// TIA Portal project "plc-automatic-manual-tank-level-control-pid" (V16)
// Vorlageprojekt für das Buch mit Zielsystem S7-1200

(* hardware
DEVICE "S7-1200-Station_1"  S7-1200 Station
   slot 0: "Baugruppenträger_0"  Rack  V1.0
   slot 1: "PLC_1"  CPU 1214C DC/DC/DC  6ES7 214-1AG40-0XB0  V4.4
   slot 2: "AQ 4x14BIT_1"  6ES7 232-4HD32-0XB0  V2.1
DEVICE "HMI_1"  KTP700 Basic PN
   slot 0: "HMI_1"  KTP700 Basic PN  6AV2 123-2GB03-0AX0  16.0.0.0
   slot 1: "HMI_RT_1"  KTP700 Basic PN  6AV2 123-2GB03-0AX0  16.0.0.0
   slot 5: "HMI_1.IE_CP_1"  PROFINET Interface  16.0.0.0
      slot 1: "PROFINET Interface_1"  PROFINET Interface
         slot 1: "Port_1"  Port
*)

// ===== PLC "PLC_1"  CPU 1214C DC/DC/DC =====

VAR_GLOBAL   // PLC tag table "Standard-Variablentabelle"
   "Seviye_Sensörü" AT %IW30 : Int;
   "Doldurma_Valfi" AT %QW30 : Int;
   "Set_Point" AT %MW32 : Int;
   "HMI_Doldurma_But" AT %M5.0 : Bool;
   "PID_Çıkış_Mem" AT %MW10 : Int;
   "HMI_OTO_MAN" AT %M5.1 : Bool;
   "HMI_Boşaltma_But" AT %M5.3 : Bool;
   "Man_Doldurma_Mem" AT %M5.4 : Bool;
   "DolVlf_Açıklık_DInt" AT %MD12 : DInt;
   "Otomatik_Start_Mem" AT %M5.5 : Bool;
   "HMI_Sıvı_Seviye" AT %MD34 : Real;
   "DolVlf_Açıklık_Yüzde_DInt" AT %MD16 : DInt;
   "Sıvı_Seviye_Mem" AT %MW38 : Int;
   "Sıvı_Seviye" AT %MD40 : Real;
   "Boşaltma_Valfi" AT %QW32 : Int;
   "Üst_Limit" AT %M5.7 : Bool;
   "Man_Boşaltma_Mem" AT %M6.0 : Bool;
   "HMI_DolVlf_Açıklık_Arttır_But" AT %M6.1 : Bool;
   "HMI_DolVlf_Açıklık_Azalt_But" AT %M6.2 : Bool;
   "HMI_BoşVlf_Açıklık_Arttır_But" AT %M6.3 : Bool;
   "HMI_BoşVlf_Açıklık_Azalt_But" AT %M6.4 : Bool;
   "DolVlf_Açıklık_Mem" AT %MW44 : Int;
   "BoşVlf_Açıklık_Mem" AT %MW46 : Int;
   "HMI_DolVlf_Açıklık_Yüzde" AT %MW20 : Int;
   "BoşVlf_Açıklık_DInt" AT %MD22 : DInt;
   "BoşVlf_Açıklık_Yüzde_DInt" AT %MD26 : DInt;
   "HMI_BoşVlf_Açıklık_Yüzde" AT %MW30 : Int;
   "Kenar_Tetikleme_1" AT %M6.5 : Bool;
   "Kenar_Tetikleme_2" AT %M6.6 : Bool;
   "Kenar_Tetikleme_3" AT %M6.7 : Bool;
   "Kenar_Tetikleme_4" AT %M7.0 : Bool;
   "DolVlf_Açıklık_Kontrol" AT %MW50 : Int;
   "HMI_Stop_But" AT %M5.2 : Bool;
   "Clock_Byte" AT %MB0 : Byte;
   "Clock_10Hz" AT %M0.0 : Bool;
   "Clock_5Hz" AT %M0.1 : Bool;
   "Clock_2.5Hz" AT %M0.2 : Bool;
   "Clock_2Hz" AT %M0.3 : Bool;
   "Clock_1.25Hz" AT %M0.4 : Bool;
   "Clock_1Hz" AT %M0.5 : Bool;
   "Clock_0.625Hz" AT %M0.6 : Bool;
   "Clock_0.5Hz" AT %M0.7 : Bool;
   "Stop_Uyarı" AT %M7.1 : Bool;
END_VAR

FUNCTION "Manuel_Çalışma" : Void   // FC1, LAD
{ S7_Optimized_Access := 'TRUE' }
VERSION : 0.1
BEGIN

REGION Network 1
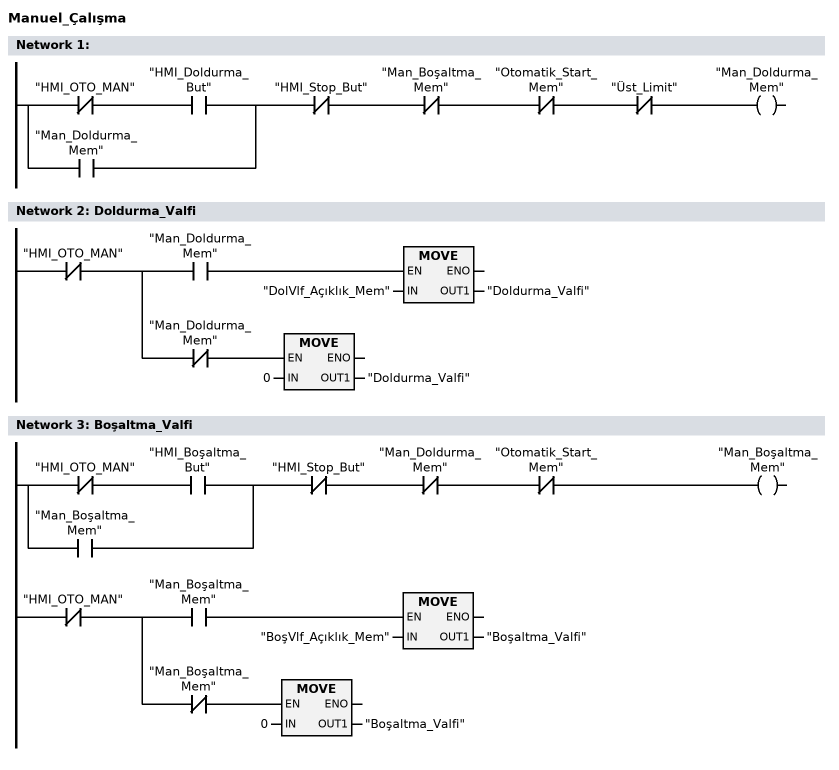
   RUNG wire#powerrail
      I_Contact( "HMI_OTO_MAN" )
      Contact( "HMI_Doldurma_But" )
      wire#w1
      I_Contact( "HMI_Stop_But" )
      I_Contact( "Man_Boşaltma_Mem" )
      I_Contact( "Otomatik_Start_Mem" )
      I_Contact( "Üst_Limit" )
      Coil( "Man_Doldurma_Mem" )
   END_RUNG
   RUNG wire#powerrail
      Contact( "Man_Doldurma_Mem" )
   END_RUNG wire#w1
   // the same network as SCL:
   "Man_Doldurma_Mem" := ((NOT "HMI_OTO_MAN" AND "HMI_Doldurma_But") OR "Man_Doldurma_Mem") AND NOT "HMI_Stop_But" AND NOT "Man_Boşaltma_Mem" AND NOT "Otomatik_Start_Mem" AND NOT "Üst_Limit";
END_REGION

REGION Network 2: Doldurma_Valfi
   RUNG wire#powerrail
      I_Contact( "HMI_OTO_MAN" )
      wire#w1
      Contact( "Man_Doldurma_Mem" )
      Move(in := "DolVlf_Açıklık_Mem", out1 => "Doldurma_Valfi")
   END_RUNG
   RUNG wire#w1
      I_Contact( "Man_Doldurma_Mem" )
      Move(in := 0, out1 => "Doldurma_Valfi")
   END_RUNG
   // the same network as SCL:
   IF NOT "HMI_OTO_MAN" AND "Man_Doldurma_Mem" THEN "Doldurma_Valfi" := "DolVlf_Açıklık_Mem"; END_IF;
   IF NOT "HMI_OTO_MAN" AND NOT "Man_Doldurma_Mem" THEN "Doldurma_Valfi" := 0; END_IF;
END_REGION

REGION Network 3: Boşaltma_Valfi
   RUNG wire#powerrail
      I_Contact( "HMI_OTO_MAN" )
      Contact( "HMI_Boşaltma_But" )
      wire#w1
      I_Contact( "HMI_Stop_But" )
      I_Contact( "Man_Doldurma_Mem" )
      I_Contact( "Otomatik_Start_Mem" )
      Coil( "Man_Boşaltma_Mem" )
   END_RUNG
   RUNG wire#powerrail
      Contact( "Man_Boşaltma_Mem" )
   END_RUNG wire#w1
   RUNG wire#powerrail
      I_Contact( "HMI_OTO_MAN" )
      wire#w2
      Contact( "Man_Boşaltma_Mem" )
      Move(in := "BoşVlf_Açıklık_Mem", out1 => "Boşaltma_Valfi")
   END_RUNG
   RUNG wire#w2
      I_Contact( "Man_Boşaltma_Mem" )
      Move(in := 0, out1 => "Boşaltma_Valfi")
   END_RUNG
   // the same network as SCL:
   "Man_Boşaltma_Mem" := ((NOT "HMI_OTO_MAN" AND "HMI_Boşaltma_But") OR "Man_Boşaltma_Mem") AND NOT "HMI_Stop_But" AND NOT "Man_Doldurma_Mem" AND NOT "Otomatik_Start_Mem";
   IF NOT "HMI_OTO_MAN" AND "Man_Boşaltma_Mem" THEN "Boşaltma_Valfi" := "BoşVlf_Açıklık_Mem"; END_IF;
   IF NOT "HMI_OTO_MAN" AND NOT "Man_Boşaltma_Mem" THEN "Boşaltma_Valfi" := 0; END_IF;
END_REGION
END_FUNCTION

FUNCTION "Otomatik_Çalışma" : Void   // FC2, LAD
{ S7_Optimized_Access := 'TRUE' }
VERSION : 0.1
BEGIN

REGION Network 1
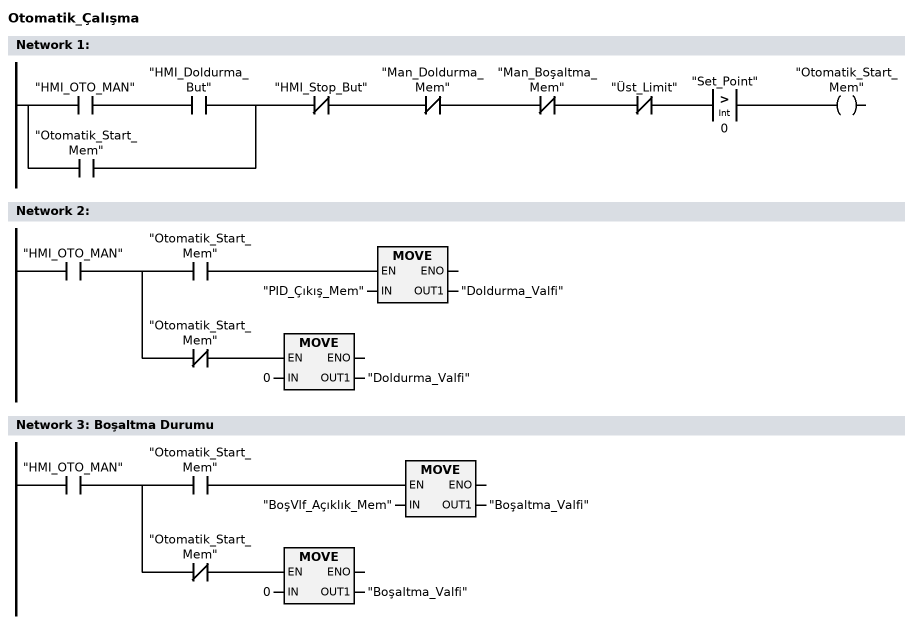
   RUNG wire#powerrail
      Contact( "HMI_OTO_MAN" )
      Contact( "HMI_Doldurma_But" )
      wire#w1
      I_Contact( "HMI_Stop_But" )
      I_Contact( "Man_Doldurma_Mem" )
      I_Contact( "Man_Boşaltma_Mem" )
      I_Contact( "Üst_Limit" )
      { S7_Templates := "SrcType := Int" } GT_Contact(in1 := "Set_Point", in2 := 0)
      Coil( "Otomatik_Start_Mem" )
   END_RUNG
   RUNG wire#powerrail
      Contact( "Otomatik_Start_Mem" )
   END_RUNG wire#w1
   // the same network as SCL:
   "Otomatik_Start_Mem" := (("HMI_OTO_MAN" AND "HMI_Doldurma_But") OR "Otomatik_Start_Mem") AND NOT "HMI_Stop_But" AND NOT "Man_Doldurma_Mem" AND NOT "Man_Boşaltma_Mem" AND NOT "Üst_Limit" AND ("Set_Point" > 0);
END_REGION

REGION Network 2
   RUNG wire#powerrail
      Contact( "HMI_OTO_MAN" )
      wire#w1
      Contact( "Otomatik_Start_Mem" )
      Move(in := "PID_Çıkış_Mem", out1 => "Doldurma_Valfi")
   END_RUNG
   RUNG wire#w1
      I_Contact( "Otomatik_Start_Mem" )
      Move(in := 0, out1 => "Doldurma_Valfi")
   END_RUNG
   // the same network as SCL:
   IF "HMI_OTO_MAN" AND "Otomatik_Start_Mem" THEN "Doldurma_Valfi" := "PID_Çıkış_Mem"; END_IF;
   IF "HMI_OTO_MAN" AND NOT "Otomatik_Start_Mem" THEN "Doldurma_Valfi" := 0; END_IF;
END_REGION

REGION Network 3: Boşaltma Durumu
   RUNG wire#powerrail
      Contact( "HMI_OTO_MAN" )
      wire#w1
      Contact( "Otomatik_Start_Mem" )
      Move(in := "BoşVlf_Açıklık_Mem", out1 => "Boşaltma_Valfi")
   END_RUNG
   RUNG wire#w1
      I_Contact( "Otomatik_Start_Mem" )
      Move(in := 0, out1 => "Boşaltma_Valfi")
   END_RUNG
   // the same network as SCL:
   IF "HMI_OTO_MAN" AND "Otomatik_Start_Mem" THEN "Boşaltma_Valfi" := "BoşVlf_Açıklık_Mem"; END_IF;
   IF "HMI_OTO_MAN" AND NOT "Otomatik_Start_Mem" THEN "Boşaltma_Valfi" := 0; END_IF;
END_REGION
END_FUNCTION

FUNCTION "MHJ-PLC-Lab-Function-S71200" : Void   // FC9000, SCL
{ S7_Optimized_Access := 'TRUE' }
VERSION : 0.1
   VAR_TEMP
      rdTimeReturn : Int;
      outputTime : DTL;
      SyncVal : Byte;
      forVal : Int;
      forVal_2 : Int;
      Value : Byte;
   END_VAR
   VAR CONSTANT
      CompVal : Byte := 16#34;
      Value_01 : Byte := 16#11;
      Value_01_DW : DWord := 16#A165_D992;
      Value_02_DW : DWord := 16#58BE_4401;
   END_VAR
BEGIN

   #Value:=PEEK(area := 16#82,
        dbNumber := 0,
        byteOffset := 511);
   #Value := #Value + 1;

   POKE(area := 16#82,
        dbNumber := 0,
        byteOffset := 511,
        value := #Value);

   POKE(area:=16#81,
        dbNumber:=0,
        byteOffset:=1016,
        value:=#Value_01_DW);
   POKE(area := 16#81,
        dbNumber := 0,
        byteOffset := 1020,
        value := #Value_02_DW);

   POKE(area := 16#81,
        dbNumber := 0,
        byteOffset := 511,
        value := B#16#00);

   FOR #forVal := 0 TO 120 DO
       FOR #forVal_2:=0 TO 10 DO
           #rdTimeReturn:=RD_SYS_T(#outputTime);
           #rdTimeReturn := WR_SYS_T(#outputTime);
           #rdTimeReturn := RD_SYS_T(#outputTime);
           #rdTimeReturn := WR_SYS_T(#outputTime);
       END_FOR;
       #SyncVal:= PEEK(area := 16#81,
                      dbNumber := 0,
                      byteOffset := 511);
       IF #SyncVal = #CompVal THEN
          GOTO M_1;
       END_IF;
   END_FOR;
   RETURN;

   M_1:
   POKE(area := 16#81,
        dbNumber := 0,
        byteOffset := 511,
        value := B#16#0);
END_FUNCTION

ORGANIZATION_BLOCK "Main"   // OB1, LAD, ProgramCycle
TITLE = "Main Program Sweep (Cycle)"
{ S7_Optimized_Access := 'TRUE' }
VERSION : 0.1
   VAR_INPUT
      Initial_Call : Bool;   // Initial call of this OB
      Remanence : Bool;   // =True, if remanent data are available
   END_VAR
   VAR_TEMP   // added for the SCL form of the ladder/FBD networks
      _w1 : Bool;
      _w2 : Bool;
   END_VAR
BEGIN

REGION Network 1: Konnektierungsbaustein für PLC-Lab
   // Im Netzwerk 1 wird der Konnektierungsbaustein für PLC-Lab aufgerufen.
   // Dieser Aufruf darf nicht entfernt werden!
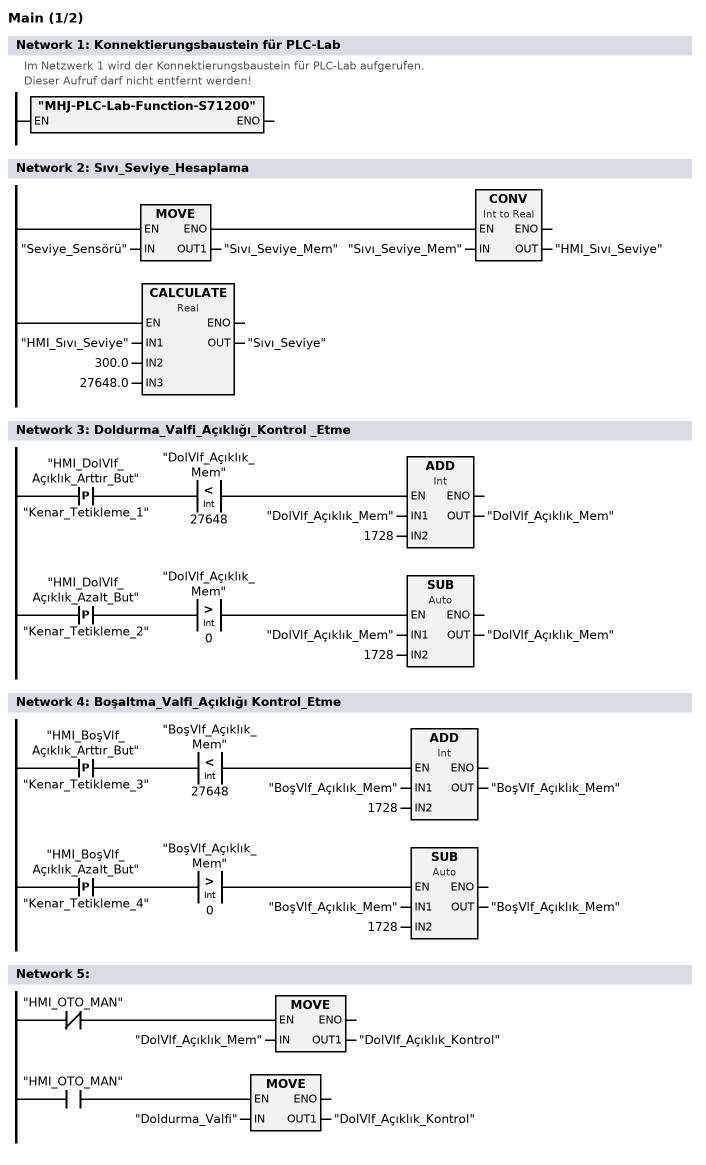
   RUNG wire#powerrail
      "MHJ-PLC-Lab-Function-S71200"()
   END_RUNG
   // the same network as SCL:
   "MHJ-PLC-Lab-Function-S71200"();
END_REGION

REGION Network 2: Sıvı_Seviye_Hesaplama
   RUNG wire#powerrail
      Move(in := "Seviye_Sensörü", out1 => "Sıvı_Seviye_Mem")
      { S7_Templates := "[SrcType := Int, DestType := Real]" } Convert(in := "Sıvı_Seviye_Mem", out => "HMI_Sıvı_Seviye")
   END_RUNG
   RUNG wire#powerrail
      { S7_Templates := "SrcType := Real"; S7_Expression := "(IN1*IN2)/IN3" } Calculate(in1 := "HMI_Sıvı_Seviye", in2 := 300.0, in3 := 27648.0, out => "Sıvı_Seviye")
   END_RUNG
   // the same network as SCL:
   "Sıvı_Seviye_Mem" := "Seviye_Sensörü";
   "HMI_Sıvı_Seviye" := INT_TO_REAL("Sıvı_Seviye_Mem");
   "Sıvı_Seviye" := ("HMI_Sıvı_Seviye"*300.0)/27648.0;
END_REGION

REGION Network 3: Doldurma_Valfi_Açıklığı_Kontrol _Etme
   RUNG wire#powerrail
      P_Contact(operand := "HMI_DolVlf_Açıklık_Arttır_But", bit := "Kenar_Tetikleme_1")
      { S7_Templates := "SrcType := Int" } LT_Contact(in1 := "DolVlf_Açıklık_Mem", in2 := 27648)
      { S7_Templates := "SrcType := Int" } Add(in1 := "DolVlf_Açıklık_Mem", in2 := 1728, out => "DolVlf_Açıklık_Mem")
   END_RUNG
   RUNG wire#powerrail
      P_Contact(operand := "HMI_DolVlf_Açıklık_Azalt_But", bit := "Kenar_Tetikleme_2")
      { S7_Templates := "SrcType := Int" } GT_Contact(in1 := "DolVlf_Açıklık_Mem", in2 := 0)
      Sub(in1 := "DolVlf_Açıklık_Mem", in2 := 1728, out => "DolVlf_Açıklık_Mem")
   END_RUNG
   // the same network as SCL:
   #_w1 := "HMI_DolVlf_Açıklık_Arttır_But" AND NOT "Kenar_Tetikleme_1";   // rising edge of "HMI_DolVlf_Açıklık_Arttır_But"
   "Kenar_Tetikleme_1" := "HMI_DolVlf_Açıklık_Arttır_But";
   IF #_w1 AND ("DolVlf_Açıklık_Mem" < 27648) THEN
       "DolVlf_Açıklık_Mem" := "DolVlf_Açıklık_Mem" + 1728;
   END_IF;
   #_w2 := "HMI_DolVlf_Açıklık_Azalt_But" AND NOT "Kenar_Tetikleme_2";   // rising edge of "HMI_DolVlf_Açıklık_Azalt_But"
   "Kenar_Tetikleme_2" := "HMI_DolVlf_Açıklık_Azalt_But";
   IF #_w2 AND ("DolVlf_Açıklık_Mem" > 0) THEN "DolVlf_Açıklık_Mem" := "DolVlf_Açıklık_Mem" - 1728; END_IF;
END_REGION

REGION Network 4: Boşaltma_Valfi_Açıklığı Kontrol_Etme
   RUNG wire#powerrail
      P_Contact(operand := "HMI_BoşVlf_Açıklık_Arttır_But", bit := "Kenar_Tetikleme_3")
      { S7_Templates := "SrcType := Int" } LT_Contact(in1 := "BoşVlf_Açıklık_Mem", in2 := 27648)
      { S7_Templates := "SrcType := Int" } Add(in1 := "BoşVlf_Açıklık_Mem", in2 := 1728, out => "BoşVlf_Açıklık_Mem")
   END_RUNG
   RUNG wire#powerrail
      P_Contact(operand := "HMI_BoşVlf_Açıklık_Azalt_But", bit := "Kenar_Tetikleme_4")
      { S7_Templates := "SrcType := Int" } GT_Contact(in1 := "BoşVlf_Açıklık_Mem", in2 := 0)
      Sub(in1 := "BoşVlf_Açıklık_Mem", in2 := 1728, out => "BoşVlf_Açıklık_Mem")
   END_RUNG
   // the same network as SCL:
   #_w1 := "HMI_BoşVlf_Açıklık_Arttır_But" AND NOT "Kenar_Tetikleme_3";   // rising edge of "HMI_BoşVlf_Açıklık_Arttır_But"
   "Kenar_Tetikleme_3" := "HMI_BoşVlf_Açıklık_Arttır_But";
   IF #_w1 AND ("BoşVlf_Açıklık_Mem" < 27648) THEN
       "BoşVlf_Açıklık_Mem" := "BoşVlf_Açıklık_Mem" + 1728;
   END_IF;
   #_w2 := "HMI_BoşVlf_Açıklık_Azalt_But" AND NOT "Kenar_Tetikleme_4";   // rising edge of "HMI_BoşVlf_Açıklık_Azalt_But"
   "Kenar_Tetikleme_4" := "HMI_BoşVlf_Açıklık_Azalt_But";
   IF #_w2 AND ("BoşVlf_Açıklık_Mem" > 0) THEN "BoşVlf_Açıklık_Mem" := "BoşVlf_Açıklık_Mem" - 1728; END_IF;
END_REGION

REGION Network 5
   RUNG wire#powerrail
      I_Contact( "HMI_OTO_MAN" )
      Move(in := "DolVlf_Açıklık_Mem", out1 => "DolVlf_Açıklık_Kontrol")
   END_RUNG
   RUNG wire#powerrail
      Contact( "HMI_OTO_MAN" )
      Move(in := "Doldurma_Valfi", out1 => "DolVlf_Açıklık_Kontrol")
   END_RUNG
   // the same network as SCL:
   IF NOT "HMI_OTO_MAN" THEN "DolVlf_Açıklık_Kontrol" := "DolVlf_Açıklık_Mem"; END_IF;
   IF "HMI_OTO_MAN" THEN "DolVlf_Açıklık_Kontrol" := "Doldurma_Valfi"; END_IF;
END_REGION

REGION Network 6: HMI_DolValf_Açıklığı_Yüzdesi
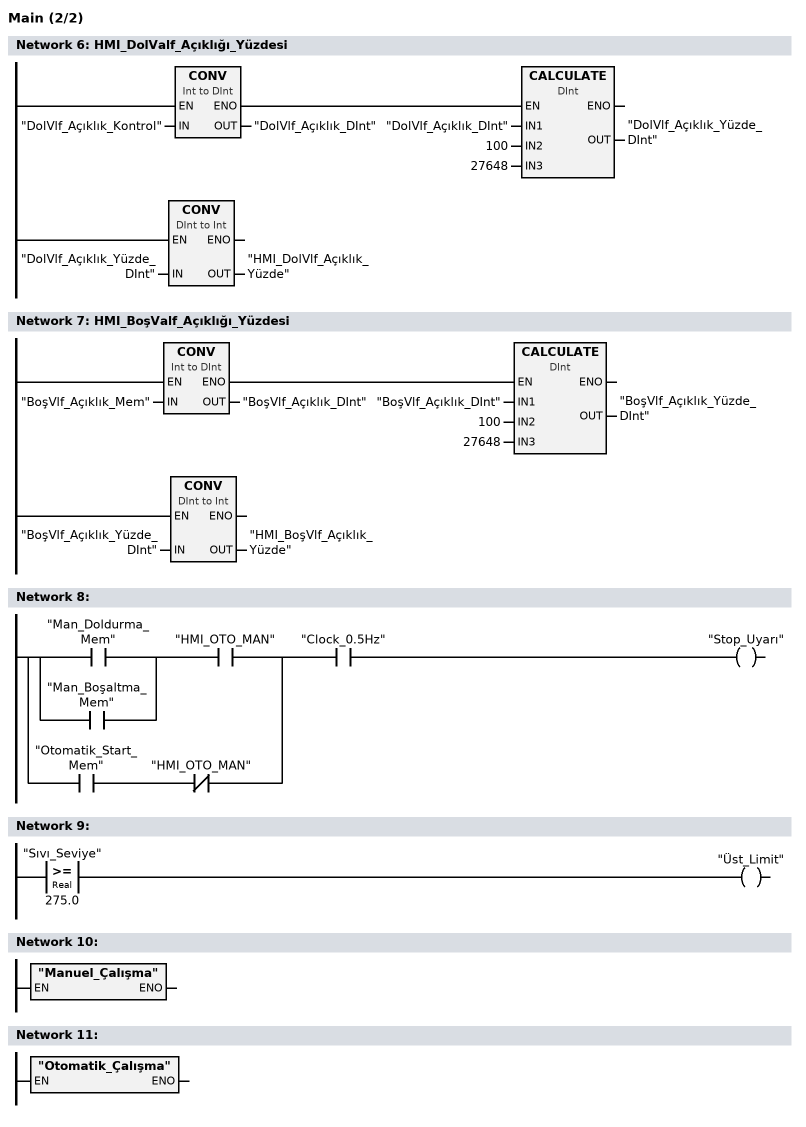
   RUNG wire#powerrail
      { S7_Templates := "[SrcType := Int, DestType := DInt]" } Convert(in := "DolVlf_Açıklık_Kontrol", out => "DolVlf_Açıklık_DInt")
      { S7_Templates := "SrcType := DInt"; S7_Expression := "(IN1*IN2)/IN3" } Calculate(in1 := "DolVlf_Açıklık_DInt", in2 := 100, in3 := 27648, out => "DolVlf_Açıklık_Yüzde_DInt")
   END_RUNG
   RUNG wire#powerrail
      { S7_Templates := "[SrcType := DInt, DestType := Int]" } Convert(in := "DolVlf_Açıklık_Yüzde_DInt", out => "HMI_DolVlf_Açıklık_Yüzde")
   END_RUNG
   // the same network as SCL:
   "DolVlf_Açıklık_DInt" := INT_TO_DINT("DolVlf_Açıklık_Kontrol");
   "DolVlf_Açıklık_Yüzde_DInt" := ("DolVlf_Açıklık_DInt"*100)/27648;
   "HMI_DolVlf_Açıklık_Yüzde" := DINT_TO_INT("DolVlf_Açıklık_Yüzde_DInt");
END_REGION

REGION Network 7: HMI_BoşValf_Açıklığı_Yüzdesi
   RUNG wire#powerrail
      { S7_Templates := "[SrcType := Int, DestType := DInt]" } Convert(in := "BoşVlf_Açıklık_Mem", out => "BoşVlf_Açıklık_DInt")
      { S7_Templates := "SrcType := DInt"; S7_Expression := "(IN1*IN2)/IN3" } Calculate(in1 := "BoşVlf_Açıklık_DInt", in2 := 100, in3 := 27648, out => "BoşVlf_Açıklık_Yüzde_DInt")
   END_RUNG
   RUNG wire#powerrail
      { S7_Templates := "[SrcType := DInt, DestType := Int]" } Convert(in := "BoşVlf_Açıklık_Yüzde_DInt", out => "HMI_BoşVlf_Açıklık_Yüzde")
   END_RUNG
   // the same network as SCL:
   "BoşVlf_Açıklık_DInt" := INT_TO_DINT("BoşVlf_Açıklık_Mem");
   "BoşVlf_Açıklık_Yüzde_DInt" := ("BoşVlf_Açıklık_DInt"*100)/27648;
   "HMI_BoşVlf_Açıklık_Yüzde" := DINT_TO_INT("BoşVlf_Açıklık_Yüzde_DInt");
END_REGION

REGION Network 8
   RUNG wire#powerrail
      Contact( "Man_Doldurma_Mem" )
      wire#w1
      Contact( "HMI_OTO_MAN" )
      wire#w2
      Contact( "Clock_0.5Hz" )
      Coil( "Stop_Uyarı" )
   END_RUNG
   RUNG wire#powerrail
      Contact( "Man_Boşaltma_Mem" )
   END_RUNG wire#w1
   RUNG wire#powerrail
      Contact( "Otomatik_Start_Mem" )
      I_Contact( "HMI_OTO_MAN" )
   END_RUNG wire#w2
   // the same network as SCL:
   "Stop_Uyarı" := ((("Man_Doldurma_Mem" OR "Man_Boşaltma_Mem") AND "HMI_OTO_MAN") OR ("Otomatik_Start_Mem" AND NOT "HMI_OTO_MAN")) AND "Clock_0.5Hz";
END_REGION

REGION Network 9
   RUNG wire#powerrail
      { S7_Templates := "SrcType := Real" } GE_Contact(in1 := "Sıvı_Seviye", in2 := 275.0)
      Coil( "Üst_Limit" )
   END_RUNG
   // the same network as SCL:
   "Üst_Limit" := "Sıvı_Seviye" >= 275.0;
END_REGION

REGION Network 10
   RUNG wire#powerrail
      "Manuel_Çalışma"()
   END_RUNG
   // the same network as SCL:
   "Manuel_Çalışma"();
END_REGION

REGION Network 11
   RUNG wire#powerrail
      "Otomatik_Çalışma"()
   END_RUNG
   // the same network as SCL:
   "Otomatik_Çalışma"();
END_REGION
END_ORGANIZATION_BLOCK

ORGANIZATION_BLOCK "Cyclic interrupt"   // OB30, LAD, CyclicInterrupt
{ S7_Optimized_Access := 'TRUE' }
VERSION : 0.1
   VAR_INPUT
      Initial_Call : Bool;   // Initial call of this OB
      Event_Count : Int;   // Events discarded
   END_VAR
BEGIN

REGION Network 1
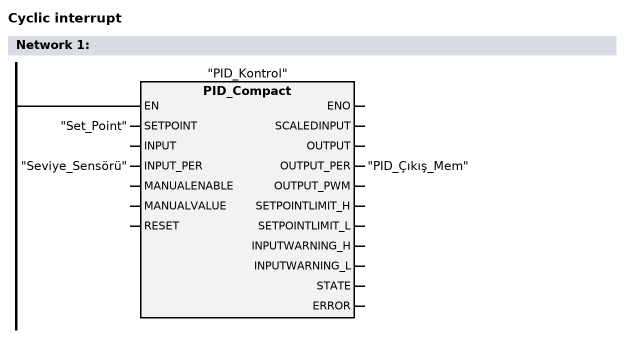
   "PID_Kontrol"(Setpoint := "Set_Point", Input_PER := "Seviye_Sensörü", Output_PER => "PID_Çıkış_Mem");   // PID_Compact
END_REGION
END_ORGANIZATION_BLOCK

(* ===== HMI "HMI_RT_1" =====
system functions are stored by id; their names below are inferred from use
connection "HMI_Connection_1": ETHERNET, SMART_S7_1200_OMS

HMI tags "Default tag table"
   "Tag_ScreenNumber" : UInt, internal
   "HMI_OTO_MAN" : Bool = PLC HMI_OTO_MAN AT %M5.1, 1 s
   "HMI_Start_But" : Bool = PLC HMI_Doldurma_But AT %M5.0, 1 s
   "Set_Point" : Int = PLC Set_Point AT %MW32, 1 s
   "Sıvı_Seviye" : Real = PLC Sıvı_Seviye AT %MD40, 1 s
   "HMI_Boşaltma_But" : Bool = PLC HMI_Boşaltma_But AT %M5.3, 1 s
   "HMI_DolVlf_Açıklık_Arttır_But" : Bool = PLC HMI_DolVlf_Açıklık_Arttır_But AT %M6.1, 1 s
   "HMI_DolVlf_Açıklık_Azalt_But" : Bool = PLC HMI_DolVlf_Açıklık_Azalt_But AT %M6.2, 1 s
   "HMI_BoşVlf_Açıklık_Arttır_But" : Bool = PLC HMI_BoşVlf_Açıklık_Arttır_But AT %M6.3, 1 s
   "HMI_BoşVlf_Açıklık_Azalt_But" : Bool = PLC HMI_BoşVlf_Açıklık_Azalt_But AT %M6.4, 1 s
   "HMI_DolVlf_Açıklık_Yüzde" : Int = PLC HMI_DolVlf_Açıklık_Yüzde AT %MW20, 1 s
   "HMI_BoşVlf_Açıklık_Yüzde" : Int = PLC HMI_BoşVlf_Açıklık_Yüzde AT %MW30, 1 s
   "HMI_Stop_But" : Bool = PLC HMI_Stop_But AT %M5.2, 1 s
   "Stop_Uyarı" : Bool = PLC Stop_Uyarı AT %M7.1, 1 s

graphic list "Graphic_list_1": 0..1 'Down_Arrow'

screen "Ana Sayfa" 800x480
   on GenerateScreen: SetTag("Tag_ScreenNumber", 1)
   Switch "Rotary_RG" at 86,108 size 80x80; CaptionText 'Switch'; TextOff '0'; TextOn '1'; PictureOff "Rotary_RG_Off_256c"; PictureOn "Rotary_RG_On_256c"
      ProcessValue <- "HMI_OTO_MAN"
   Bar "Bar_1" at 609,90 size 116x273; MinimumValue 0; MaximumValue 300
      ProcessValue <- "Sıvı_Seviye"
   TextField "Text field_1" at 272,16 size 266x43; Text 'TANK KONTROL PANELİ'
   IOField "I/O field_1" at 486,120 size 75x35; FormatPattern 999
      ProcessValue <- "Set_Point"
   TextField "Text field_2" at 66,87 size 135x18; Text 'MANUEL | OTOMATİK'
   TextField "Text field_3" at 484,306 size 77x18; Text 'SIVI SEVİYE'
   IOField "I/O field_2" at 484,260 size 75x35; FormatPattern 999.99
      ProcessValue <- "Sıvı_Seviye"
   TextField "Text field_4" at 444,167 size 156x20; Text 'SIVI SEVİYE SET DEĞERİ'
   IOField "I/O field_3" at 297,167 size 50x30; FormatPattern 999
      ProcessValue <- "HMI_DolVlf_Açıklık_Yüzde"
   TextField "Text field_5" at 297,123 size 119x32; Text 'DOLDURMA VALFİ AÇIKLIĞI'
   TextField "Text field_6" at 561,126 size 14x23; Text 'L'
   TextField "Text field_7" at 559,267 size 14x23; Text 'L'
   TextField "Text field_8" at 349,172 size 24x23; Text '%'
   Button "Button_1" at 235,105 size 50x50; TextOff 'Text'; PictureOff "Up_Arrow"
      on Press: SetBit("HMI_DolVlf_Açıklık_Arttır_But")
      on Release: ResetBit("HMI_DolVlf_Açıklık_Arttır_But")
      Appearance <- "HMI_OTO_MAN"
   Button "Button_2" at 235,172 size 50x50; TextOff 'Text'; PictureOff "Down_Arrow"
      on Press: SetBit("HMI_DolVlf_Açıklık_Azalt_But")
      on Release: ResetBit("HMI_DolVlf_Açıklık_Azalt_But")
      Appearance <- "HMI_OTO_MAN"
   Button "Button_3" at 235,245 size 50x50; TextOff 'Text'; PictureOff "Up_Arrow"
      on Press: SetBit("HMI_BoşVlf_Açıklık_Arttır_But")
      on Release: ResetBit("HMI_BoşVlf_Açıklık_Arttır_But")
   Button "Button_4" at 235,306 size 50x50; TextOff 'Text'; PictureOff "Down_Arrow"
      on Press: SetBit("HMI_BoşVlf_Açıklık_Azalt_But")
      on Release: ResetBit("HMI_BoşVlf_Açıklık_Azalt_But")
   IOField "I/O field_4" at 299,306 size 50x30; FormatPattern 999
      ProcessValue <- "HMI_BoşVlf_Açıklık_Yüzde"
   TextField "Text field_9" at 299,263 size 116x32; Text 'BOŞALTMA VALFİ AÇIKLIĞI'
   TextField "Text field_10" at 349,310 size 24x23; Text '%'
   Button "Button_5" at 65,344 size 120x40; TextOff 'STOP'
      on Press: SetBit("HMI_Stop_But")
      on Release: ResetBit("HMI_Stop_But")
   Button "Button_7" at 66,230 size 120x40; TextOff 'DOLDUR'
      on Press: SetBit("HMI_Start_But")
      on Release: ResetBit("HMI_Start_But")
   Button "Button_8" at 65,287 size 120x40; TextOff 'BOŞALT'
      on Press: SetBit("HMI_Boşaltma_But")
      on Release: ResetBit("HMI_Boşaltma_But")
   TextField "Text field_11" at 38,192 size 179x23; Text 'SİSTEMİ STOP EDİN !'
      Visibility <- "Stop_Uyarı"
   Softkey "Softkey_F8" at 0,0 size 0x0; SoftkeyImage "Right_Arrow"
      on KeyDown: ActivateScreen("Trend_Ekranı", 0)

screen "Trend_Ekranı" 800x480
   TrendView "Trend view_1" at 83,65 size 637x345
   TextField "Text field_1" at 272,23 size 240x23; Text 'SIVI SEVİYE ANALİZ EKRANI'
   Softkey "Softkey_F1" at 0,0 size 0x0; SoftkeyImage "Left_Arrow"
      on KeyDown: ActivateScreen("Ana Sayfa", 0)
*)